(* CODESYS project HowToUse_MIC7001_baselib.2020.0205.1.project

Project tree, tasks and I/O mapping:
  Device : Changsha-Cyber-MI-linux, Changsha Cyber-MI Co., Ltd., version 3.5.10.40
    application Application
      libraries: Standard, * (System); SysFile, 3.5.15.0 (System); SysTypes2 Interfaces, * (System); SysShm, * (System); CAA Mathematics, * (CAA Technical Workgroup); SysTime, 3.5.9.0 (System); CAA Types Extern, 3.5.13.0 (CAA Technical Workgroup); CAA DTUtil Extern, 3.5.12.0 (CAA Technical Workgroup); Util, * (System); MIC7001 base library, 0.76 (Cyber-MI.com); TCP, 3.5.15.0 (3S - Smart Software Solutions GmbH); CAA Net Base Services, 3.5.15.0 (CAA Technical Workgroup)
      task c_MainTask (cyclic, interval 10 ms, priority 20) calls prg_heartbeat, prg_data2file, prg_retain
      Enums/
        data type ERROR
        data type MQTT_STATE
        data type UDP_STATE_1
      data type UDP_STATE
      programs/
        program prg_heartbeat [ST]
        program prg_data2file [ST]
        program prg_retain [ST]
      Functions/
        function Enable_120ohm_can0 [ST]
        function write_num_to_file [ST]
        function read_num_from_file [ST]
        function Enable_120ohm_can1 [ST]
        function Disable_120ohm_can0 [ST]
        function Disable_120ohm_can1 [ST]
        function Set_piv01 [ST]
        function Set_piv23 [ST]
        function set_ip [ST]
        function set_wifi_passwd [ST]
        function read_iccid [ST]
        function read_ip [ST]
        function read_sn [ST]
        function read_wifi_passwd [ST]
        function read_work_mins [ST]
        function read_location [ST]
      heartbeat/
        function fn_cyber_layer1 [ST]
        function fn_cyber_layer2 [ST]
        function fn_cyber_heartBeat [ST]
        function fn_sn_str_to_byte [ST]
        function Iccid_to_bytes [ST]
    SoftMotion General Axis Pool
    IoDrvMIC7001 : IoDrvMIC7001, Cyber-MI, version 19.1.1
        output Application.prg_heartbeat.running_light : BOOL  // LED_run
        unmapped channels: Ai00@C16, Ai01@C28, Ai02@C17, Ai03@C29, Ai04@C30, Ai05@C19, Ai06@C31, Ai07@C20, Ai08@C18, Ai09@D18, Ai10@D20, Ai11@D31, Ai12@D19, Ai13@D30, Ai14@D29, Ai15@D17, Ai16@D28, Ai17@D16, Ai18-Do00@C25, Ai19-Do01@C24, Ai20-Do02@C13, Ai21-Do03@C01, Ai22-Do04@C03, Ai23-Do05@C04, Ai24-Do06@C05, Ai25-Do07@C06, Ai26-Do08@C08, Ai27-Do09@C09, Ai28-Do10@C10, Ai29-Do11@C11, Ai30-Do12@D34, Ai31-Do13@D35, Ai32-Do14@D23, Ai33-Do15@D12, Ai34-Do16@D10, Ai35-Do17@D09, Ai36-Do18@D08, Ai37-Do19@D07, Ai38-Do20@D05, Ai39-Do21@D04,
          Ai40-Do22@D03, Ai41-Do23@D02, Ai42-Do24@C23, Ai43-Do25@C35, Ai44-Do26@D24, Ai45-Do27@D13, Ai46-Ao00@C22, Ai47-Ao01@D14, Ai48_Pi02, Ai49_Out5V, Ai50_VCC, Ai51_VCC_L, Ai52_VCC_R, Ai53_Pwm-i0, Ai54_Pwm-i1, Ai55_Pwm-i2, Ai56_Pwm-i3, Ai57_CPU-T, Ai58_G-x, Ai59_G-y, Ai60_G-z, Ai61-reserved, Ai62-IO-cntr, Ai63-CDS-cntr, Di00-Ai00@C16, Di01-Ai01@C28, Di02-Ai02@C17, Di03-Ai03@C29, Di04-Ai04@C30, Di05-Ai05@C19, Di06-Ai06@C31, Di07-Ai07@C20, Di08-Ai08@C18, Di09-Ai09@D18, Di10-Ai10@D20, Di11-Ai11@D31, Di12-Ai12@D19, Di13-Ai13@D30, Di14-Ai14@D29, Di15-Ai15@D17,
          Di16-Ai16@D28, Di17-Ai17@D16, Di18-Ai18@C25, Di19-Ai19@C24, Di20-Ai20@C13, Di21-Ai21@C01, Di22-Ai22@C03, Di23-Ai23@C04, Di24-Ai24@C05, Di25-Ai25@C06, Di26-Ai26@C08, Di27-Ai27@C09, Di28-Ai28@C10, Di29-Ai29@C11, Di30-Ai30@D34, Di31-Ai31@D35, Di32-Ai32@D23, Di33-Ai33@D12, Di34-Ai34@D10, Di35-Ai35@D09, Di36-Ai36@D08, Di37-Ai37@D07, Di38-Ai38@D05, Di39-Ai39@D04, Di40-Ai40@D03, Di41-Ai41@D02, Di42-Ai42@C23, Di43-Ai43@C35, Di44-Ai44@D24, Di45-Ai45@D13, Di46-Ai46@C22, Di47-Ai47@D14, Di48-Pi00@C15, Di49-Pi01@C14, Di50-Pi02@D22, Di51-Pi03@D21, Di52-reserved, Di53-reserved, Di54-reserved, Di55-reserved,
          Di56-reserved, Di57-reserved, Di58-reserved, Di59-reserved, Di60-reserved, Di61-reserved, Di62-reserved, Di63-reserved, Pi00-Di48@C15, Pi01-Di49@C14, Pi02-Di50@D22, Pi03-Di51@D21, Do00-Ai18@C25, Do01-Ai19@C24, Do02-Ai20@C13, Do03-Ai21@C01, Do04-Ai22@C03, Do05-Ai23@C04, Do06-Ai24@C05, Do07-Ai25@C06, Do08-Ai26@C08, Do09-Ai27@C09, Do10-Ai28@C10, Do11-Ai29@C11, Do12-Ai30@D34, Do13-Ai31@D35, Do14-Ai32@D23, Do15-Ai33@D12, Do16-Ai34@D10, Do17-Ai35@D09, Do18-Ai36@D08, Do19-Ai37@D07, Do20-Ai38@D05, Do21-Ai39@D04, Do22-Ai40@D03, Do23-Ai41@D02, Do24-Ai42@C23, Do25-Ai43@C35, Do26-Ai44@D24, Do27-Ai45@D13,
          Do28-Pwmi00@C33, Do29-Pwmi01@C34, Do30-Pwmi02@D25, Do31-Pwmi03@D26, PWM00@C25, PWM01@C24, PWM02@C13, PWM03@C01, PWM04@C03, PWM05@C04, PWM06@C05, PWM07@C06, PWM08@C08, PWM09@C09, PWM10@C10, PWM11@C11, PWM12@D34, PWM13@D35, PWM14@D23, PWM15@D12, PWM16@D10, PWM17@D09, PWM18@D08, PWM19@D07, PWM20@D05, PWM21@D04, PWM22@D03, PWM23@D02, PWM24@C23, PWM25@C35, PWM26@D24, PWM27@D13, PWM28-Pwmi00@C33, PWM29-Pwmi01@C34, PWM30-Pwmi02@D25, PWM31-Pwmi03@D26, PWM_I_0@C33, PWM_I_1@C34, PWM_I_2@D25, PWM_I_3@D26,
          Ao00-Ai46@C22, Ao01-Ai47@D14, LED_err, LED_usr, ctrl_ai_raw, ctrl_adjust, ctrl_adj0, ctrl_adj1, ctrl_adj2, ctrl_adj3, disable_5V
  libraries: VisuSymbols, 3.5.10.0 (System)
  5ce3da45-db07-42e7-a21c-a00fff4ed8f6|C:\Users\zhou\p01.bmp
  5ce3da45-db07-42e7-a21c-a00fff4ed8f6|C:\working\p01.bmp
  5ce3da45-db07-42e7-a21c-a00fff4ed8f6|C:\working\file.bmp
  text list GlobalTextList
*)

// Device/Application/UDP_STATE
TYPE UDP_STATE :
(
	INIT := 0, 	(* first State. Connections are set up *)
	SEND,		(* Send messages *)
	READ,		(* Receive messages *)
	ERROR		(* Prepare to reset connections *)
);
END_TYPE

// Device/Application/Enums/ERROR
{attribute 'qualified_only'}
//{attribute 'conditionalshow'}
//{attribute 'conditionalshow' := 'SomeText'}
//{attribute 'hide'}
TYPE ERROR : (NO_ERROR, TIME_OUT); END_TYPE

// Device/Application/Enums/MQTT_STATE
{attribute 'qualified_only'}
{attribute 'strict'}
TYPE MQTT_STATE :
(
	INIT := 0,
	CONN_SEND,
	CONN_RECV,
	READY,
	SEND,
	RECV,
	ERROR
);
END_TYPE

// Device/Application/Enums/UDP_STATE_1
TYPE UDP_STATE_1 :
(
	INIT := 0, 	(* first State. Connections are set up *)
	SEND,		(* Send messages *)
	READ,		(* Receive messages *)
	ERROR		(* Prepare to reset connections *)
);
END_TYPE

// Device/Application/programs/prg_heartbeat
PROGRAM prg_heartbeat
VAR_OUTPUT
	lock_state :INT := 0;
	unlock_state :INT := 0;
	lock_unlock_level :INT := 0;
	delay_time :INT := 0;
END_VAR

VAR
	is_inited :BOOL := FALSE;
	eSTATE			: UDP_STATE; (* 状态转换变量 *)
	
	myIP		: NBS.IP_ADDR; (* MIC7001本身的IP地址 *)
	myPort		: UINT; (* MIC7001用于通信的端口 *)
	IPSend		: NBS.IP_ADDR; (* 对方的IP地址 *)
	PortSend	: UINT; (* 对方的端口 *)

	sToSend			: STRING; (* 待发送数据 *)
	sReceived		: STRING; (* 接收数据 *)
	
	UDPPeer			: NBS.UDP_Peer; (* FB UDP Peer *)
	UDPSend			: NBS.UDP_Send; (* FB UDP Send *)
	UDPReceive		: NBS.UDP_Receive; (* FB UDP Receive *)
	Peer			: CAA.HANDLE; (* Handle to the peer connection *)

	size :CAA.SIZE;	
	Writebuffer: 			ARRAY[1..200] OF BYTE;
	Readbuffer: 			ARRAY[0..1499] OF BYTE;
	ReadbufferStr: STRING;
	atcState :INT := 0;
	
	writeUdpState :INT := 0;
	readUdpState :INT := 0;
	
	i :INT;
	count :INT := 0;
	
	rtc_fb: RTC;
	dtu_set_dt_fb: dtu.SetDateAndTime;
	
	
	//server_ip:STRING := '47.107.240.29';
	//server_port:UINT := 34567;
	
	server_ip:STRING := '47.107.240.29';
    server_port:UINT := 20861;
	
	is_read :BOOL := FALSE;
	read_count :INT := 0;
	readFileState :INT := 0;
	ton_fb :TON;
	iccid_read_buffer :STRING;
	position :INT := -1;
	new_date:DT;
	iStat :UINT := 0;
	lac : STRING(4) := '0000';
	ci : STRING(4) := '0000';
	lenHearBeat:UINT;
	dataHearBeat:ARRAY[0..255] OF BYTE;
	ton_hb:ton; //heartbeat timer 
	bReturn:BOOL;
	lenLayer2:UINT;
	dataLayer2:ARRAY[0..255] OF BYTE;
	lenLayer1:UINT;
	lenRecvLayer1:UINT := 1500;
	dataLayer1:ARRAY[0..255] OF BYTE;
	bSN :ARRAY[0..6] OF BYTE;
	sub_str:STRING(8);
	num :UINT;
	lenHeartBeat: UINT;
	sn: STRING;
	work_time: DINT;
	dataIndex :UINT := 0;
	cntr_lac:UINT := 0;
	cntr_iccid:UINT := 0;
	cntr_recv:UINT := 0;
	dataLayern:ARRAY[1..255] OF BYTE;
	recv_size :CAA.SIZE;
	
	/// 辅助变量 
	xSend			: BOOL;
	sTmp1			: STRING;
	xEnable			: BOOL;	
	gprs_serial :CAA.HANDLE;
	
	ton_run:TON;
	running_light:BOOL := FALSE;
END_VAR

//运行灯每秒闪烁一次
ton_run(in := NOT ton_run.Q, pt := T#500MS);
IF ton_run.Q THEN
	running_light := NOT running_light;
END_IF

CASE iStat OF
0:
	xEnable:= TRUE;  //用于启动最下方的第70行的UDPPeer
	// 建立连接后马上转到发送状态
	IF UDPPeer.xActive THEN 
		eSTATE:= UDP_STATE.send;
	ELSIF UDPPeer.xError THEN
		eSTATE:= UDP_STATE.ERROR;
	END_IF
	
	//UDPPeer.ipAddr.sAddr := '192.168.2.253';
	UDPPeer.ipAddr.sAddr := '0.0.0.0';
	UDPPeer.uiPort := 12345;  //port of MIC7001
	IPSend.sAddr := server_ip;
	iStat := 2;
	
2:
	IF NOT read_iccid(ADR(iccid_read_buffer)) THEN
		iccid_read_buffer := 'iccid_null';		
	END_IF;
	iStat := 10;
	
10: //read sn
	IF NOT read_sn(ADR(sn)) THEN 
		sn := 'sn_null';
	END_IF
	
	iStat := 15;
	
15:
	read_location(ADR(lac), ADR(ci));
	iStat := 30;
30:
	work_time := read_work_mins();
	iStat := 100;
	
100:   //定时等待
	ton_fb(IN := TRUE, PT := T#10S);
	IF (ton_fb.Q) THEN
		ton_fb(IN := FALSE, PT := T#10S);
		iStat := 200;  //发送心跳
	ELSE
		iStat := 300; //发送实时数据	
	END_IF
	
200:
	bReturn := fn_cyber_heartBeat(	  //填充第三层：心跳帧
						lac_str := lac, 
						cid_str := ci, 
						ccid_str := iccid_read_buffer, 
						mins := work_time, 
						clientCode := 6,   //hengtian 95
						machineCode := 5,  //挖掘机
						pLenOut := ADR(lenHearBeat), 
						pDataOut := ADR(dataHearBeat)
	);
	
	IF NOT bReturn THEN
		RETURN;
	END_IF;

	dataIndex := dataIndex + 1;
	bReturn := fn_cyber_layer2( //填充第二层，数据层
						dataType := 1,
						paraId := 0,
						dataIndex := dataIndex,
						ver := 1,
						res1 := 0,
						LenIn := lenHearBeat,
						pDataIn := ADR(dataHearBeat),
						pLenOut := ADR(lenLayer2),
						pDataOut := ADR(dataLayer2)
	);
				
	IF NOT bReturn THEN
		RETURN;
	END_IF;

	bSN := fn_sn_str_to_byte(sn);
	bReturn := fn_cyber_layer1(    //填充第一层，设备层
						sn := ADR(bSN),
						ver := 1,
						lenIn := lenLayer2,
						pDataIn := ADR(dataLayer2),
						pLenOut := ADR(lenLayer1),
						pDataOut := ADR(dataLayer1)
	);
	
	IF NOT bReturn THEN
		RETURN;
	ELSE
		UDPSend(xExecute := FALSE);
		iStat := 500;
	END_IF;
	
300:  //sending realtime data  here
	//UDPSend(some realtime data as need);
	iStat := 100;
	
500:
	UDPSend(xExecute := TRUE, hPeer := Peer, ipAddr := IPSend, uiPort := server_port, szSize := lenLayer1, pDAta := ADR(dataLayer1));
	IF UDPSend.xDone THEN
		UDPSend(xExecute := FALSE);
		iStat := 600; 
	END_IF
	
	IF UDPSend.xError THEN  
		UDPSend(xExecute := FALSE);
		iStat := 30; 
	END_IF
	
	
600:
	UDPReceive(xEnable := UDPPeer.xActive, hPeer := Peer, szSize := SIZEOF(Readbuffer), pData := ADR(Readbuffer));
	IF UDPReceive.xReady THEN  //接收到数据
	 	recv_size := UDPReceive.szCount;
		UDPReceive(xEnable := FALSE);
		iStat := 30; //read mins and lca again
		IF recv_size = 26 THEN
			lock_state := BYTE_TO_INT(Readbuffer[20]);
			unlock_state := BYTE_TO_INT(Readbuffer[21]);
			lock_unlock_level := BYTE_TO_INT(Readbuffer[22]);
			delay_time := BYTE_TO_INT(Readbuffer[23]);
		END_IF
	ELSE
		cntr_recv := cntr_recv + 1;
		IF cntr_recv > 2000 THEN
			cntr_recv := 0;
			iStat := 30;
		END_IF
	END_IF
	
	IF UDPReceive.xError THEN  //接收错误
		UDPReceive(xEnable := FALSE);
		recv_size := 0;
		iStat := 30; //read mins and lca again
	END_IF
END_CASE

//保持每个周期调用，维护与对方的连接关系本地端口的接收状态
UDPPeer(xEnable:= xEnable, hPeer=> Peer);
RETURN;

END_PROGRAM

// Device/Application/Functions/read_iccid
FUNCTION read_iccid : BOOL
VAR_INPUT
	iccid: POINTER TO STRING;
END_VAR

VAR
	hFile: RTS_IEC_HANDLE;
	udiOpenError: RTS_IEC_RESULT;
	udiReadError: RTS_IEC_RESULT;
	i :INT;
	iTemp: UDINT;
	udiPos: UDINT;
	str_size: __XWORD;
	udiByteRead: LWORD;

	len_of_line: INT;
	len_of_number :INT;
	magicNumber:REAL;
	check_sum:REAL:= 0;
	temp_num:REAL;
END_VAR

read_iccid := FALSE;

//检测文件是否存在
hFile := sysfileopen(szFile := '/userapp/iccid.txt', am := sysfile.AM_READ, pResult:= ADR(udiOpenError));
IF hFile = RTS_INVALID_HANDLE	THEN  //文件不存在
	RETURN;
END_IF
//文件存在，开始读取内容
udiPos := SysFileSetPos(hFile:=hFile, ulOffset := 0);
udiByteRead := sysfile.SysFileRead(hfile := hFile,pbyBuffer := iccid, ulSize := 32, pResult := ADR(udiReadError));
IF udiByteRead < 4 THEN  //读取失败
	sysfile.SysFileClose(hFile := hFile);
	RETURN;
END_IF

sysfile.SysFileClose(hFile := hFile);
read_iccid := TRUE;

END_FUNCTION

// Device/Application/Functions/read_sn
FUNCTION read_sn : BOOL
VAR_INPUT
	sn: POINTER TO STRING;
END_VAR

VAR
	hFile: RTS_IEC_HANDLE;
	udiOpenError: RTS_IEC_RESULT;
	udiReadError: RTS_IEC_RESULT;
	i :INT;
	iTemp: UDINT;
	udiPos: UDINT;
	str_size: __XWORD;
	udiByteRead: LWORD;

	len_of_line: INT;
	len_of_number :INT;
	magicNumber:REAL;
	check_sum:REAL:= 0;
	temp_num:REAL;
END_VAR

read_sn := FALSE;

//检测文件是否存在
hFile := sysfileopen(szFile := '/userapp/sn.txt', am := sysfile.AM_READ, pResult:= ADR(udiOpenError));
IF hFile = RTS_INVALID_HANDLE	THEN  //文件不存在
	RETURN;
END_IF
//文件存在，开始读取内容
udiPos := SysFileSetPos(hFile:=hFile, ulOffset := 0);
udiByteRead := sysfile.SysFileRead(hfile := hFile,pbyBuffer := sn, ulSize := 32, pResult := ADR(udiReadError));
IF udiByteRead < 4 THEN  //读取失败
	sysfile.SysFileClose(hFile := hFile);
	RETURN;
END_IF
sysfile.SysFileClose(hFile := hFile);
read_sn := TRUE;

END_FUNCTION

// Device/Application/Functions/read_location
FUNCTION read_location : BOOL
VAR_INPUT
	lac:POINTER TO STRING;
	ci:POINTER TO STRING;
END_VAR

VAR
	hFile: RTS_IEC_HANDLE;
	udiOpenError: RTS_IEC_RESULT;
	udiReadError: RTS_IEC_RESULT;
	i :INT;
	iTemp: UDINT;
	udiPos: UDINT;
	str_size: __XWORD;
	udiByteRead: LWORD;

	len_of_line: INT;
	len_of_number :INT;
	magicNumber:REAL;
	check_sum:REAL:= 0;
	temp_num:REAL;	
END_VAR

read_location := FALSE;
lac^ := '0000';
ci^ := '0000';

//检测文件是否存在
hFile := sysfileopen(szFile := '/userapp/laccid.txt', am := sysfile.AM_READ, pResult:= ADR(udiOpenError));
IF hFile = RTS_INVALID_HANDLE	THEN  //文件不存在
	RETURN;
END_IF

//文件存在，开始读取内容
udiPos := SysFileSetPos(hFile:=hFile, ulOffset := 0);
udiByteRead := sysfile.SysFileRead(hfile := hFile,pbyBuffer := lac, ulSize := 32, pResult := ADR(udiReadError));
IF udiByteRead < 4 THEN  //读取失败
	sysfile.SysFileClose(hFile := hFile);
	RETURN;
END_IF
sysfile.SysFileClose(hFile := hFile);

hFile := sysfileopen(szFile := '/userapp/cid.txt', am := sysfile.AM_READ, pResult:= ADR(udiOpenError));
IF hFile = RTS_INVALID_HANDLE	THEN  //文件不存在
	RETURN;
END_IF

//文件存在，开始读取内容
udiPos := SysFileSetPos(hFile:=hFile, ulOffset := 0);
udiByteRead := sysfile.SysFileRead(hfile := hFile,pbyBuffer := ci, ulSize := 32, pResult := ADR(udiReadError));
IF udiByteRead < 4 THEN  //读取失败
	sysfile.SysFileClose(hFile := hFile);
	RETURN;
END_IF
sysfile.SysFileClose(hFile := hFile);

read_location := TRUE;

END_FUNCTION

// Device/Application/Functions/read_work_mins
FUNCTION read_work_mins : DINT;
VAR_INPUT
END_VAR

VAR
	time_file_name :STRING := '/userapp/r_mins.txt';
	hFile: RTS_IEC_HANDLE;
	udiOpenError: RTS_IEC_RESULT;
	udiReadError: RTS_IEC_RESULT;

	udiPos: UDINT;
	str_size: __XWORD;
	udiByteRead: LWORD;
	read_buf:STRING;

END_VAR

read_work_mins := 0;

//检测文件是否存在
hFile := sysfileopen(szFile := time_file_name, am := sysfile.AM_READ, pResult:= ADR(udiOpenError));
IF hFile = RTS_INVALID_HANDLE	THEN  //文件不存在
	RETURN;
END_IF

//文件存在，开始读取内容
udiPos := SysFileSetPos(hFile:=hFile, ulOffset := 0);
udiByteRead := sysfile.SysFileRead(hfile := hFile,pbyBuffer := ADR(read_buf), ulSize := 32, pResult := ADR(udiReadError));
sysfile.SysFileClose(hFile := hFile);

read_work_mins := ANY_TO_DINT(read_buf);

END_FUNCTION

// Device/Application/heartbeat/fn_cyber_heartBeat
FUNCTION fn_cyber_heartBeat : bool
VAR_INPUT
	lac_str:STRING(4);
	cid_str:STRING(4);
	ccid_str:STRING(21);
	mins:UDINT;
	clientCode:UINT;
	machineCode:UINT;
	pLenOut:POINTER TO UINT;
	pDataOut:POINTER TO BYTE;
END_VAR
VAR
	index: UINT;
	data_uint: UINT;
	data_byte_array:ARRAY[0..9] OF BYTE;
	i: INT;
END_VAR

fn_cyber_heartBeat := FALSE;

index := 0;
data_uint := STRING_TO_UINT(concat('16#',lac_str));
pDataOut[index] := ANY_TO_BYTE(data_uint/256);
index := index + 1;

pDataOut[index] := ANY_TO_BYTE(data_uint MOD 256);
index := index + 1;

data_uint := STRING_TO_UINT(concat('16#',cid_str));
pDataOut[index] := ANY_TO_BYTE(data_uint/256);
index := index + 1;

pDataOut[index] := ANY_TO_BYTE(data_uint MOD 256);
index := index + 1;

data_byte_array := Iccid_to_bytes(ccid_str);
FOR i := 0 TO 9 DO
	pDataOut[index] := data_byte_array[i];
	index := index + 1;
END_FOR

pDataOut[index] := ANY_TO_BYTE(mins/256/256/256);
index := index + 1;

pDataOut[index] := ANY_TO_BYTE(mins/256/256);
index := index + 1;

pDataOut[index] := ANY_TO_BYTE(mins/256);
index := index + 1;

pDataOut[index] := ANY_TO_BYTE(mins);
index := index + 1;

pDataOut[index] := ANY_TO_BYTE(clientCode/256);
index := index + 1;

pDataOut[index] := ANY_TO_BYTE(clientCode);
index := index + 1;

pDataOut[index] := ANY_TO_BYTE(machineCode/256);
index := index + 1;

pDataOut[index] := ANY_TO_BYTE(machineCode);
index := index + 1;

pLenOut^ := index;

fn_cyber_heartBeat := TRUE;

END_FUNCTION

// Device/Application/heartbeat/Iccid_to_bytes
FUNCTION Iccid_to_bytes : ARRAY[0..9] OF BYTE
VAR_INPUT
	iccd :STRING;
END_VAR
VAR
	iccid_code :ARRAY[0..9] OF BYTE;
	
	byteHigh :BYTE := 0;
	byteLow :BYTE := 0;
	dstLen :INT := 0;
	
	srcIndex :INT := 0;
	bytesIndex :INT := 0;
	sub_str:STRING(32);
END_VAR

dstLen := len(iccd) / 2;

sub_str := iccd;
FOR bytesIndex := 0 TO dstLen - 1 DO
	iccid_code[bytesIndex] := BYTE_TO_BCD(STRING_TO_BYTE(left(sub_str,2)));	
	sub_str := delete(sub_str,2,1);
END_FOR

Iccid_to_bytes := iccid_code;

END_FUNCTION

// Device/Application/heartbeat/fn_cyber_layer2
FUNCTION fn_cyber_layer2 : bool
VAR_INPUT
	dataType : BYTE := 0;
	paraId :BYTE := 0;
	dataIndex : UINT := 0;
	ver :BYTE := 1;
	res1 :BYTE := 0;
	LenIn :UINT := 0;
	pDataIn :POINTER TO BYTE;
	pLenOut :POINTER TO UINT;
	pDataOut :POINTER TO BYTE;
END_VAR
VAR
	i:UINT:= 0;
	index:UINT := 0;
END_VAR

fn_cyber_layer2 := FALSE;

index := 0;
pDataOut[index] := dataType;
index := index + 1;

pDataOut[index] := paraId;
index := index + 1;

pDataOut[index] := ANY_TO_BYTE(dataIndex/256);
index := index + 1;

pDataOut[index] := ANY_TO_BYTE(dataIndex MOD 256);
index := index + 1;

pDataOut[index] := ver;
index := index + 1;

pDataOut[index] := res1;
index := index + 1;

pDataOut[index] := ANY_TO_BYTE(LenIn/256);
index := index + 1;

pDataOut[index] := ANY_TO_BYTE(LenIn MOD 256);
index := index + 1;

FOR i := 0 TO LenIn-1 DO
	pDataOut[index] := pDataIn[i];
	index := index + 1;
END_FOR

pLenOut^ := index;

fn_cyber_layer2 := TRUE;
RETURN;

END_FUNCTION

// Device/Application/heartbeat/fn_sn_str_to_byte
FUNCTION fn_sn_str_to_byte : ARRAY[0..6] OF BYTE
VAR_INPUT
	sn:STRING(16);
END_VAR
VAR
	i: INT;
	bSN: ARRAY[0..6] OF BYTE;
	sub_str: STRING(255);
	num: UINT;
	bcd: UINT;
END_VAR

// 1.2 12
sub_str := mid(sn, 2, 4);
bcd := STRING_TO_UINT(sub_str);
bcd := (bcd / 10) *16 + (bcd MOD 10);
bSN[0] := UINT_TO_BYTE(bcd);

// 1.3 34
sub_str := mid(sn, 2, 6);
bcd := STRING_TO_UINT(sub_str);
bcd := (bcd / 10) *16 + (bcd MOD 10);
bSN[1] := UINT_TO_BYTE(bcd);

// 1.4 56
sub_str := mid(sn, 2, 8);
bcd := STRING_TO_UINT(sub_str);
bcd := (bcd / 10) *16 + (bcd MOD 10);
bSN[2] := UINT_TO_BYTE(bcd);

// 1.5 78
sub_str := mid(sn, 2, 10);
bcd := STRING_TO_UINT(sub_str);
bcd := (bcd / 10) *16 + (bcd MOD 10);
bSN[3] := UINT_TO_BYTE(bcd);

// 1.6 1234
sub_str := mid(sn, 2, 12);
bcd := STRING_TO_UINT(sub_str);
bcd := (bcd / 10) *16 + (bcd MOD 10);
bSN[4] := UINT_TO_BYTE(bcd);

sub_str := mid(sn, 2, 14);
bcd := STRING_TO_UINT(sub_str);
bcd := (bcd / 10) *16 + (bcd MOD 10);
bSN[5] := UINT_TO_BYTE(bcd);

fn_sn_str_to_byte := bSN;

END_FUNCTION

// Device/Application/heartbeat/fn_cyber_layer1
FUNCTION fn_cyber_layer1 : bool
VAR_INPUT
	sn:POINTER TO BYTE;
	ver:BYTE := 0;
	lenIn:UINT := 0;
	pDataIn:POINTER TO BYTE;
	pLenOut:POINTER TO UINT ;
	pDataOut: POINTER TO BYTE;
END_VAR
VAR
	i:UINT;
	index:UINT;
	checksum:UINT;
END_VAR

fn_cyber_layer1 := FALSE;

index := 0;
checksum := 0;
FOR i := 0 TO 8 DO
	pDataOut[index] := sn[i];
	index := index+1;
	checksum := checksum + sn[i];
END_FOR

pDataOut[index] := ver;
index := index+1;
checksum := checksum + ver;

pDataOut[index] := ANY_TO_BYTE(lenIn/256);
index := index+1;
checksum := checksum + ANY_TO_BYTE(lenIn/256);

pDataOut[index] := ANY_TO_BYTE(lenIn MOD 256);
index := index+1;
checksum := checksum + ANY_TO_BYTE(lenIn MOD 256);

FOR i := 0 TO lenIn-1 DO
	pDataOut[index] := pDataIn[i];
	index := index+1;	
	checksum := checksum + pDataIn[i];
END_FOR

pDataOut[index] := ANY_TO_BYTE(checksum/256);
index := index+1;

pDataOut[index] := ANY_TO_BYTE(checksum MOD 256);
index := index+1;

pLenOut^ := index;

fn_cyber_layer1 := TRUE;

END_FUNCTION

// Device/Application/programs/prg_data2file
PROGRAM prg_data2file
VAR
	data:ARRAY[0..MIC7001_base.Constants.FILE_DATA_MAX] OF REAL;
	data2file :MIC7001_base.FB_DATA2FILE;
	
	init:BOOL:= FALSE;
	hFile: RTS_IEC_HANDLE := RTS_INVALID_HANDLE;
	udiOpenError: RTS_IEC_RESULT;
	udiWriteError: RTS_IEC_RESULT;
	
	start_save:BOOL := FALSE;
	i:UINT := 0;
	cntr :real := 1.23;
END_VAR


data2file.xEnable := TRUE;
cntr := cntr + 1;

data[0] := 123.456;
FOR i := 1 TO 255 DO
	data[i] := data[0]*(cntr+6);
END_FOR

data2file(data := data, length := 255, interval := T#300MS, filedir := '/userdata/', maxsize_m := 100);

END_PROGRAM

// Device/Application/programs/prg_retain
PROGRAM prg_retain
VAR
	myRetain:mic7001_base.FB_RETAIN;
	inited:BOOL := FALSE;
	//retain 变量, 建议放在全局变量列表 gvl中
	g_retain:ARRAY[0..mic7001_base.Constants.RETAIN_NUM_MAX] OF DINT;
END_VAR

//步骤一：初始化默认值,如果读取文件失败，则使用默认值作为当前参数
IF NOT inited THEN  //上电执行一次，设置retain变量的缺省值
	myRetain.default_val[0] := 123;
	myRetain.default_val[1] := 456;
	myRetain.default_val[2] := 789;
	// .....
	myRetain.default_val[87] := 321;
	myRetain.default_val[88] := 654;
	
	myRetain(value := g_retain);
	
	inited := TRUE;
END_IF


//步骤二：执行功能块，处理参数的保存和读取
myRetain(value := g_retain);

//步骤三：在其它任务中直接使用 g_retain[] 作为retain变量

END_PROGRAM

// Device/Application/Functions/Enable_120ohm_can0
FUNCTION Enable_120ohm_can0 : BOOL
VAR_INPUT
END_VAR
VAR
	filename:STRING(32) := '/userapp/can0_r_en.txt';
END_VAR

Enable_120ohm_can0 := FALSE;

IF read_num_from_file(filename := filename) < 1 THEN
	Enable_120ohm_can0 := write_num_to_file(filename := filename, num := 1);
END_IF

RETURN;

END_FUNCTION

// Device/Application/Functions/read_num_from_file
FUNCTION read_num_from_file : dint
VAR_INPUT
	filename:STRING(32);
END_VAR
VAR
	hFile: RTS_IEC_HANDLE := 0;
	udiOpenError: RTS_IEC_RESULT;
	udiReadError: RTS_IEC_RESULT;
	rdbuf:STRING(32);	
END_VAR

read_num_from_file := -1;

hFile := sysfileopen(szFile := filename, am := sysfile.AM_READ, pResult:= ADR(udiOpenError));
IF hFile = RTS_INVALID_HANDLE THEN
	RETURN;
END_IF

SysFileSetPos(hFile:=hFile, ulOffset := 0);
sysfileread(hFile := hFile, pbyBuffer := ADR(rdbuf), ulSize := SIZEOF(rdbuf), pResult := ADR(udiReadError));
sysfileClose(hFile);

read_num_from_file := ANY_TO_DINT(rdbuf);
RETURN;

END_FUNCTION

// Device/Application/Functions/write_num_to_file
FUNCTION write_num_to_file : BOOL
VAR_INPUT
	filename:STRING(32);
	num:DINT;
END_VAR
VAR
	hFile: RTS_IEC_HANDLE := 0;
	udiOpenError: RTS_IEC_RESULT;
	udiWriteError: RTS_IEC_RESULT;
	wrbuf:STRING(32);
END_VAR

write_num_to_file := FALSE;

hFile := sysfileopen(szFile := filename, am := sysfile.AM_WRITE, pResult:= ADR(udiOpenError));
IF hFile = RTS_INVALID_HANDLE THEN
	RETURN;
END_IF

wrbuf := ANY_TO_STRING(num);
wrbuf := concat(wrbuf, '$n');
SysFileSetPos(hFile:=hFile, ulOffset := 0);
sysfilewrite(hFile := hFile, pbyBuffer := ADR(wrbuf), ulSize := len(wrbuf), pResult := ADR(udiWriteError));
sysfileClose(hFile);

write_num_to_file := TRUE;

RETURN;

END_FUNCTION

// Device/Application/Functions/Enable_120ohm_can1
FUNCTION Enable_120ohm_can1 : BOOL
VAR_INPUT
END_VAR
VAR
	filename:STRING(32) := '/userapp/can1_r_en.txt';
END_VAR

Enable_120ohm_can1 := FALSE;

IF read_num_from_file(filename := filename) < 1 THEN
	Enable_120ohm_can1 := write_num_to_file(filename := filename, num := 1);
END_IF

RETURN;

END_FUNCTION

// Device/Application/Functions/Disable_120ohm_can0
FUNCTION Disable_120ohm_can0 : BOOL
VAR_INPUT
END_VAR
VAR
	filename:STRING(32) := '/userapp/can0_r_en.txt';
	num :DINT;
END_VAR

Disable_120ohm_can0 := FALSE;

num := read_num_from_file(filename := filename);
IF  NOT (num = 0)  THEN
	Disable_120ohm_can0 := write_num_to_file(filename := filename, num := 0);
END_IF

RETURN;

END_FUNCTION

// Device/Application/Functions/Disable_120ohm_can1
FUNCTION Disable_120ohm_can1 : BOOL
VAR_INPUT
END_VAR
VAR
	filename:STRING(32) := '/userapp/can1_r_en.txt';
	num :DINT;
END_VAR

Disable_120ohm_can1 := FALSE;

num := read_num_from_file(filename := filename);
IF  NOT (num = 0)  THEN
	Disable_120ohm_can1 := write_num_to_file(filename := filename, num := 0);
END_IF

RETURN;

END_FUNCTION

// Device/Application/Functions/Set_piv01
FUNCTION Set_piv01 : BOOL
VAR_INPUT
	piv_mv:DINT := 10000;  // default: 10V
END_VAR
VAR
	filename:STRING(32) := '/userapp/piv01_mv.txt';
END_VAR

Set_piv01 := FALSE;

IF read_num_from_file(filename := filename) <> piv_mv THEN
	Set_piv01 := write_num_to_file(filename := filename, num := piv_mv);
END_IF

RETURN;

END_FUNCTION

// Device/Application/Functions/Set_piv23
FUNCTION Set_piv23 : BOOL
VAR_INPUT
	piv_mv:DINT := 10000;  // default: 10V
END_VAR
VAR
	filename:STRING(32) := '/userapp/piv23_mv.txt';
END_VAR

Set_piv23 := FALSE;

IF read_num_from_file(filename := filename) <> piv_mv THEN
	Set_piv23 := write_num_to_file(filename := filename, num := piv_mv);
END_IF

RETURN;

END_FUNCTION

// Device/Application/Functions/set_ip
FUNCTION set_ip : BOOL
VAR_INPUT
	ip: POINTER TO STRING;
END_VAR
VAR
	hFile: RTS_IEC_HANDLE;
	udiOpenError: RTS_IEC_RESULT;
	udiReadError: RTS_IEC_RESULT;
	udiWriteError: RTS_IEC_RESULT;
	i :INT;
	iTemp: UDINT;
	udiPos: UDINT;
	str_size: __XWORD;
	udiByteRead: UDINT;
	length:DINT;
	
	len_of_line: INT;
	len_of_number :INT;
	magicNumber:REAL;
	check_sum:REAL:= 0;
	temp_num:REAL;
	udiByteWrite: LWORD;
END_VAR


set_ip := FALSE;

hFile := sysfileopen(szFile := '/userapp/ipaddr.txt', am := sysfile.AM_WRITE, pResult := ADR(udiOpenError));
IF hFile = RTS_INVALID_HANDLE THEN //创建文件失败
	RETURN;
END_IF

length := LEN(ip);
udiPos := SysFileSetPos(hFile:=hFile, ulOffset:=0);	
udiByteWrite := sysfile.SysFileWrite(hFile := hFile,pbyBuffer := ip,ulSize := length, pResult := ADR(udiWriteError));
IF udiByteWrite = 0 THEN
	sysfile.SysFileClose(hFile := hFile);
	RETURN;
END_IF
sysfile.SysFileClose(hFile := hFile);
set_ip := TRUE;
RETURN;

END_FUNCTION

// Device/Application/Functions/set_wifi_passwd
FUNCTION set_wifi_passwd : BOOL
VAR_INPUT
	passwd: POINTER TO STRING;
	len:DINT;
END_VAR
VAR
	hFile: RTS_IEC_HANDLE;
	udiOpenError: RTS_IEC_RESULT;
	udiReadError: RTS_IEC_RESULT;
	udiWriteError: RTS_IEC_RESULT;
	i :INT;
	iTemp: UDINT;
	udiPos: UDINT;
	str_size: __XWORD;
	udiByteRead: UDINT;

	len_of_line: INT;
	len_of_number :INT;
	magicNumber:REAL;
	check_sum:REAL:= 0;
	temp_num:REAL;
	udiByteWrite: LWORD;
END_VAR


set_wifi_passwd := FALSE;

hFile := sysfileopen(szFile := '/userapp/wifi_passwd.txt', am := sysfile.AM_WRITE, pResult := ADR(udiOpenError));
IF hFile = RTS_INVALID_HANDLE THEN //创建文件失败
	RETURN;
END_IF

udiPos := SysFileSetPos(hFile:=hFile, ulOffset:=0);	
udiByteWrite := sysfile.SysFileWrite(hFile := hFile,pbyBuffer := passwd,ulSize := len, pResult := ADR(udiWriteError));
IF udiByteWrite = 0 THEN
	sysfile.SysFileClose(hFile := hFile);
	RETURN;
END_IF

sysfile.SysFileClose(hFile := hFile);
set_wifi_passwd := TRUE;
RETURN;

END_FUNCTION

// Device/Application/Functions/read_ip
FUNCTION read_ip : BOOL
VAR_INPUT
	ip: POINTER TO STRING;
END_VAR

VAR
	hFile: RTS_IEC_HANDLE;
	udiOpenError: RTS_IEC_RESULT;
	udiReadError: RTS_IEC_RESULT;
	i :INT;
	iTemp: UDINT;
	udiPos: UDINT;
	str_size: __XWORD;
	udiByteRead: LWORD;

	len_of_line: INT;
	len_of_number :INT;
	magicNumber:REAL;
	check_sum:REAL:= 0;
	temp_num:REAL;
END_VAR

read_ip := FALSE;

//检测文件是否存在
hFile := sysfileopen(szFile := '/userapp/ipaddr.txt', am := sysfile.AM_READ, pResult:= ADR(udiOpenError));
IF hFile = RTS_INVALID_HANDLE	THEN  //文件不存在
	RETURN;
END_IF
//文件存在，开始读取内容
udiPos := SysFileSetPos(hFile:=hFile, ulOffset := 0);
udiByteRead := sysfile.SysFileRead(hfile := hFile,pbyBuffer := ip, ulSize := 32, pResult := ADR(udiReadError));
IF udiByteRead < 4 THEN  //读取失败
	sysfile.SysFileClose(hFile := hFile);
	RETURN;
END_IF
sysfile.SysFileClose(hFile := hFile);
read_ip := TRUE;

END_FUNCTION

// Device/Application/Functions/read_wifi_passwd
FUNCTION read_wifi_passwd : BOOL
VAR_INPUT
	passwd: POINTER TO STRING;
END_VAR

VAR
	hFile: RTS_IEC_HANDLE;
	udiOpenError: RTS_IEC_RESULT;
	udiReadError: RTS_IEC_RESULT;
	i :INT;
	iTemp: UDINT;
	udiPos: UDINT;
	str_size: __XWORD;
	udiByteRead: LWORD;

	len_of_line: INT;
	len_of_number :INT;
	magicNumber:REAL;
	check_sum:REAL:= 0;
	temp_num:REAL;
END_VAR

read_wifi_passwd := FALSE;

//检测文件是否存在
hFile := sysfileopen(szFile := '/userapp/wifi_passwd.txt', am := sysfile.AM_READ, pResult:= ADR(udiOpenError));
IF hFile = RTS_INVALID_HANDLE	THEN  //文件不存在
	RETURN;
END_IF
//文件存在，开始读取内容
udiPos := SysFileSetPos(hFile:=hFile, ulOffset := 0);
udiByteRead := sysfile.SysFileRead(hfile := hFile,pbyBuffer := passwd, ulSize := 32, pResult := ADR(udiReadError));
IF udiByteRead < 4 THEN  //读取失败
	sysfile.SysFileClose(hFile := hFile);
	RETURN;
END_IF
sysfile.SysFileClose(hFile := hFile);
read_wifi_passwd := TRUE;

END_FUNCTION
